// TIA Portal V20 export
FUNCTION_BLOCK "FB_ActControl"   // FB45, SCL
{ S7_Optimized_Access := 'TRUE' }
// stored: MemoryReserve 100, SetENOAutomatically false
   VAR_INPUT
      iStartSeqCond : Bool;   // Start Sequence Conditions
      iJobReq : Bool;   // Job Request - From Main
      iShuttleModeAutoPos : Bool;   // Load/Unload Manu Pos. Reached - Param
      iShuttleModeAutoPosSetPoint : LReal;   // Load/Unload Manu Pos. Setpoint - Param
      iShuttleModeSemiAutoPos : Bool;   // Load/Unload Manu Pos. Reached - Param
      iShuttleModeSemiAutoPosSetPoint : LReal;   // Load/Unload Manu Pos. Setpoint - Param
      iShuttleMoving : Bool;   // Shuttle is moving - From FB_LoaderAxis
      iShuttleInPos : Bool;   // Shuttle pos. reached - From FB_LoaderAxis
      iModeAutoPosCondition : Bool;
      iModeSemiAutoPosCondition : Bool;
      iNoStopCondition : Bool;
      iOperatorCycleRestart : Bool;
      iNC_Stopped : Bool;
      iNC_Running : Bool;
      iMissingPart : Bool;
      iExtraPart : Bool;
      iPLC_DateAndTime : DTL;
      iStepPause : Bool;
   END_VAR
   VAR_OUTPUT
      oShuttleStartReq { ExternalAccessible := 'False'; ExternalVisible := 'False'; ExternalWritable := 'False'} : Bool;   // Shuttle Start Order - To FB_LoaderAxis
      oShuttlePosSetPoint { ExternalAccessible := 'False'; ExternalVisible := 'False'; ExternalWritable := 'False'} : Real;   // Shuttle Position Setpoint - To FB_LoaderAxis
      oStopNC_Req : Bool;
      oRestartNC_Req : Bool;
      oRestartStep : Bool;
      oContinuationStep : Bool;
      oMsgMissingPart : Bool;
      oMsgExtraPart : Bool;
   END_VAR
   VAR
      sCurrent_Step_NB : Int;   // Active Step Number
      sCheck_Step_Condition : Bool;
      sOneStepForward : Bool;
      sRTOneStepForward : R_TRIG;
      sOneStepMode { S7_SetPoint := 'True'} : Bool;
      sStepForward : Bool;
      sInterface : "UDT_SequenceInterface";
      sShuttleStartReq { ExternalAccessible := 'False'; ExternalVisible := 'False'; ExternalWritable := 'False'} : Bool;
      sShuttlePosSetPoint { ExternalAccessible := 'False'; ExternalVisible := 'False'; ExternalWritable := 'False'} : Real;
      sStopNC_Req : Bool;
      sRestartNC_Req : Bool;
      sRestartStep : Bool;
      sContinuationStep : Bool;
      sMsgMissingPart : Bool;
      sMsgExtraPart : Bool;
      sHistory : Struct
         Activation : Bool;
         Steps : Array[0..99] of Int;
         Date_Time : Array[0..99] of DTL;
      END_STRUCT;
      StepText : "FB_GetTextErrorCode";
   END_VAR
   VAR_TEMP
      tIndex : Int;   // Index
   END_VAR
   VAR CONSTANT
      S00_INIT : Int := 0;
      S10_CHECK_ACT_CTRL_OPTION : Int := 10;
      S20_SHUTTLE_TO_STOP_CYCLE_POS_START_REQ : Int := 20;
      S30_SHUTTLE_TO_STOP_CYCLE_POS_REACHED : Int := 30;
      S40_STOP_CYCLE : Int := 40;
      S50_WAIT_OPERATOR_RESTART : Int := 50;
      S60_NC_RESTART : Int := 60;
      S70_UPDATE_NEXT_STEP : Int := 70;
      S120_SHUTTLE_TO_EXT_LOAD_UNLOAD_POS_START_REQ : Int := 120;
      S130_SHUTTLE_TO_EXT_LOAD_UNLOAD_POS_REACHED : Int := 130;
      S140_STOP_CYCLE : Int := 140;
      S150_WAIT_OPERATOR_RESTART : Int := 150;
      S160_NC_RESTART : Int := 160;
      S170_UPDATE_NEXT_STEP : Int := 170;
      S270_UPDATE_NEXT_STEP : Int := 270;
      S295_JOB_DONE : Int := 295;
   END_VAR
   // StepText.sCode_error[0].ErrorCode := 0;
   // StepText.sCode_error[1].ErrorCode := 10;
   // StepText.sCode_error[2].ErrorCode := 20;
   // StepText.sCode_error[3].ErrorCode := 30;
   // StepText.sCode_error[4].ErrorCode := 40;
   // StepText.sCode_error[5].ErrorCode := 50;
   // StepText.sCode_error[6].ErrorCode := 60;
   // StepText.sCode_error[7].ErrorCode := 70;
   // StepText.sCode_error[8].ErrorCode := 80;
   // StepText.sCode_error[9].ErrorCode := 90;
   // StepText.sCode_error[10].ErrorCode := 95;
BEGIN
   REGION Description header 
       //==================================================================================
       // POSALUX Swiss SA / (C) Copyright 2025
       //----------------------------------------------------------------------------------
       // Title: FB_ActControl
       // Comment/Function: 
       // Author: Fabien WALDT
       // Engineering: TIA Portal v17
       //----------------------------------------------------------------------------------
       // Change log table:
       // Version  | Date     | Expert in charge | Changes applied
       // ---------|----------|------------------|-----------------------------------------
       // 00.00.01 | 20250527 | WFA              | First released version
       // =================================================================================
   END_REGION

   REGION Define condition to start
       IF #iStartSeqCond THEN
           #sInterface.SequenceReleased := TRUE;
       ELSE
           // Standard sequencer controls
           #sInterface.SequenceReleased := FALSE;
           #sCurrent_Step_NB := #S00_INIT;
           #sInterface.SequenceRun := FALSE;
           #sInterface.JobDone := FALSE;
           #sCheck_Step_Condition := FALSE;

           // Dedicated sequencer controls
           #sShuttleStartReq := FALSE;
           #sShuttlePosSetPoint := 0.0;
           #sStopNC_Req := FALSE;
           #sRestartNC_Req := FALSE;
           #sRestartStep := FALSE;
           #sContinuationStep := FALSE;


           // Add specifics controls 
       END_IF;

       // Reset interface error
       IF #sInterface.Reset THEN
           #sInterface.Error := FALSE;
       END_IF;

       // Reset start when axis in position
       IF #iShuttleInPos THEN
           #sShuttleStartReq := FALSE;
       END_IF;

       // One step forward
       #sRTOneStepForward.CLK := #sOneStepForward;
       #sRTOneStepForward();
       #sStepForward := (NOT #sOneStepMode OR (#sOneStepMode AND #sRTOneStepForward.Q)) AND NOT #iStepPause;
       #sOneStepForward := FALSE;

       // Action only true in dedicated steps
       #sStopNC_Req := FALSE;
       #sRestartNC_Req := FALSE;
   END_REGION

   REGION Sequence Function
       CASE #sCurrent_Step_NB OF
           #S00_INIT:
               REGION S00 INIT
                   #sCheck_Step_Condition := TRUE;
                   #sMsgMissingPart := FALSE;
                   #sMsgExtraPart := FALSE;
               END_REGION
           #S10_CHECK_ACT_CTRL_OPTION:
               REGION S10_CHECK_ACT_CTRL_OPTION
                   #sCheck_Step_Condition := TRUE;
               END_REGION
           #S20_SHUTTLE_TO_STOP_CYCLE_POS_START_REQ:
               REGION S20_SHUTTLE_TO_STOP_CYCLE_POS_START_REQ
                   #sShuttleStartReq := NOT #iShuttleModeAutoPos;
                   #sShuttlePosSetPoint := LREAL_TO_REAL(#iShuttleModeAutoPosSetPoint);
                   #sCheck_Step_Condition := TRUE;
               END_REGION
           #S30_SHUTTLE_TO_STOP_CYCLE_POS_REACHED:
               REGION S30_SHUTTLE_TO_STOP_CYCLE_POS_REACHED
                   #sCheck_Step_Condition := TRUE;
               END_REGION
           #S40_STOP_CYCLE:
               REGION S40_STOP_CYCLE
                   #sStopNC_Req := TRUE;
                   #sMsgMissingPart := #iMissingPart;
                   #sMsgExtraPart := #iExtraPart;
                   #sCheck_Step_Condition := TRUE;
               END_REGION
           #S50_WAIT_OPERATOR_RESTART:
               REGION S50_WAIT_OPERATOR_RESTART
                   #sCheck_Step_Condition := TRUE;
               END_REGION
           #S60_NC_RESTART:
               REGION S60_NC_RESTART
                   #sRestartNC_Req := TRUE;
                   #sCheck_Step_Condition := TRUE;
               END_REGION
           #S70_UPDATE_NEXT_STEP:
               REGION S70_UPDATE_NEXT_STEP
                   #sRestartStep := TRUE;
                   #sContinuationStep := FALSE;
                   #sCheck_Step_Condition := TRUE;
               END_REGION

           #S120_SHUTTLE_TO_EXT_LOAD_UNLOAD_POS_START_REQ:
               REGION S120_SHUTTLE_TO_EXT_LOAD_UNLOAD_POS_START_REQ
                   #sShuttleStartReq := NOT #iShuttleModeSemiAutoPos;
                   #sShuttlePosSetPoint := LREAL_TO_REAL(#iShuttleModeSemiAutoPosSetPoint);
                   #sCheck_Step_Condition := TRUE;
               END_REGION
           #S130_SHUTTLE_TO_EXT_LOAD_UNLOAD_POS_REACHED:
               REGION S130_SHUTTLE_TO_EXT_LOAD_UNLOAD_POS_REACHED
                   #sCheck_Step_Condition := TRUE;
               END_REGION
           #S140_STOP_CYCLE:
               REGION S140_STOP_CYCLE
                   #sStopNC_Req := TRUE;
                   #sMsgMissingPart := #iMissingPart;
                   #sMsgExtraPart := #iExtraPart;
                   #sCheck_Step_Condition := TRUE;
               END_REGION
           #S150_WAIT_OPERATOR_RESTART:
               REGION S150_WAIT_OPERATOR_RESTART
                   #sCheck_Step_Condition := TRUE;
               END_REGION
           #S160_NC_RESTART:
               REGION S160_NC_RESTART
                   #sRestartNC_Req := TRUE;
                   #sCheck_Step_Condition := TRUE;
               END_REGION
           #S170_UPDATE_NEXT_STEP:
               REGION S170_UPDATE_NEXT_STEP
                   #sRestartStep := TRUE;
                   #sContinuationStep := FALSE;
                   #sCheck_Step_Condition := TRUE;
               END_REGION

           #S270_UPDATE_NEXT_STEP:
               REGION S270_UPDATE_NEXT_STEP
                   #sRestartStep := FALSE;
                   #sContinuationStep := TRUE;
                   #sCheck_Step_Condition := TRUE;
               END_REGION

           #S295_JOB_DONE:
               REGION S295_JOB_DONE
                   #sInterface.JobDone := TRUE;
                   #sCheck_Step_Condition := TRUE;
               END_REGION
           ELSE:
               #sInterface.Error := TRUE;
       END_CASE;
   END_REGION

   REGION Sequence Next Step Condition
       IF #sCheck_Step_Condition THEN
           CASE #sCurrent_Step_NB OF
               #S00_INIT:
                   REGION S00 INIT
                       IF #sInterface.SequenceReleased AND #iJobReq THEN
                           #sCurrent_Step_NB := #S10_CHECK_ACT_CTRL_OPTION;
                           #sInterface.SequenceRun := TRUE;
                           #sCheck_Step_Condition := FALSE;
                       ELSE
                           #sInterface.SequenceRun := FALSE;
                       END_IF;
                   END_REGION
               #S10_CHECK_ACT_CTRL_OPTION:
                   REGION S10_CHECK_ACT_CTRL_OPTION
                       IF #sInterface.SequenceReleased AND #sStepForward AND #iModeAutoPosCondition AND NOT #iModeSemiAutoPosCondition AND NOT #iNoStopCondition THEN
                           #sCurrent_Step_NB := #S20_SHUTTLE_TO_STOP_CYCLE_POS_START_REQ;
                           #sCheck_Step_Condition := FALSE;
                       ELSIF #sInterface.SequenceReleased AND #sStepForward AND NOT #iModeAutoPosCondition AND #iModeSemiAutoPosCondition AND NOT #iNoStopCondition THEN
                           #sCurrent_Step_NB := #S120_SHUTTLE_TO_EXT_LOAD_UNLOAD_POS_START_REQ;
                           #sCheck_Step_Condition := FALSE;
                       ELSIF #sInterface.SequenceReleased AND #sStepForward AND NOT #iModeAutoPosCondition AND NOT #iModeSemiAutoPosCondition AND #iNoStopCondition THEN
                           #sCurrent_Step_NB := #S270_UPDATE_NEXT_STEP;
                           #sCheck_Step_Condition := FALSE;
                       END_IF;
                   END_REGION
               #S20_SHUTTLE_TO_STOP_CYCLE_POS_START_REQ:
                   REGION S20_SHUTTLE_TO_STOP_CYCLE_POS_START_REQ
                       IF #sInterface.SequenceReleased AND #sStepForward AND (#iShuttleMoving OR #iShuttleModeAutoPos) THEN
                           #sCurrent_Step_NB := #S30_SHUTTLE_TO_STOP_CYCLE_POS_REACHED;
                           #sCheck_Step_Condition := FALSE;
                       END_IF;
                   END_REGION
               #S30_SHUTTLE_TO_STOP_CYCLE_POS_REACHED:
                   REGION S30_SHUTTLE_TO_STOP_CYCLE_POS_REACHED
                       IF #sInterface.SequenceReleased AND #sStepForward AND NOT #sShuttleStartReq AND #iShuttleModeAutoPos THEN
                           #sCurrent_Step_NB := #S40_STOP_CYCLE;
                           #sCheck_Step_Condition := FALSE;
                       END_IF;
                   END_REGION
               #S40_STOP_CYCLE:
                   REGION S40_STOP_CYCLE
                       IF #sInterface.SequenceReleased AND #sStepForward AND #iNC_Stopped THEN
                           #sCurrent_Step_NB := #S50_WAIT_OPERATOR_RESTART;
                           #sCheck_Step_Condition := FALSE;
                       END_IF;
                   END_REGION
                   #S50_WAIT_OPERATOR_RESTART:
                       REGION S50_WAIT_OPERATOR_RESTART
                           IF #sInterface.SequenceReleased AND #sStepForward AND #iOperatorCycleRestart THEN
                               #sCurrent_Step_NB := #S60_NC_RESTART;
                               #sCheck_Step_Condition := FALSE;
                           END_IF;
                       END_REGION
                   #S60_NC_RESTART:
                       REGION S60_NC_RESTART
                           IF #sInterface.SequenceReleased AND #sStepForward AND #iNC_Running THEN
                               #sCurrent_Step_NB := #S70_UPDATE_NEXT_STEP;
                               #sCheck_Step_Condition := FALSE;
                           END_IF;
                       END_REGION
                   #S70_UPDATE_NEXT_STEP:
                       REGION S70_UPDATE_NEXT_STEP
                           IF #sInterface.SequenceReleased AND #sStepForward AND "AlwaysTRUE" THEN
                               #sCurrent_Step_NB := #S295_JOB_DONE;
                               #sCheck_Step_Condition := FALSE;
                           END_IF;
                       END_REGION

                   #S120_SHUTTLE_TO_EXT_LOAD_UNLOAD_POS_START_REQ:
                       REGION S120_SHUTTLE_TO_EXT_LOAD_UNLOAD_POS_START_REQ
                           IF #sInterface.SequenceReleased AND #sStepForward AND (#iShuttleMoving OR #iShuttleModeSemiAutoPos) THEN
                               #sCurrent_Step_NB := #S130_SHUTTLE_TO_EXT_LOAD_UNLOAD_POS_REACHED;
                               #sCheck_Step_Condition := FALSE;
                           END_IF;
                       END_REGION
                   #S130_SHUTTLE_TO_EXT_LOAD_UNLOAD_POS_REACHED:
                       REGION S130_SHUTTLE_TO_EXT_LOAD_UNLOAD_POS_REACHED
                           IF #sInterface.SequenceReleased AND #sStepForward AND NOT #sShuttleStartReq AND #iShuttleModeSemiAutoPos THEN
                               #sCurrent_Step_NB := #S140_STOP_CYCLE;
                               #sCheck_Step_Condition := FALSE;
                           END_IF;
                       END_REGION
                   #S140_STOP_CYCLE:
                       REGION S140_STOP_CYCLE
                           IF #sInterface.SequenceReleased AND #sStepForward AND #iNC_Stopped THEN
                               #sCurrent_Step_NB := #S150_WAIT_OPERATOR_RESTART;
                               #sCheck_Step_Condition := FALSE;
                           END_IF;
                       END_REGION
                       #S150_WAIT_OPERATOR_RESTART:
                           REGION S150_EXCHANGE_EXT_LOADER_IN_PROGRESS
                               IF #sInterface.SequenceReleased AND #sStepForward AND #iOperatorCycleRestart THEN
                                   #sCurrent_Step_NB := #S160_NC_RESTART;
                                   #sCheck_Step_Condition := FALSE;
                               END_IF;
                           END_REGION
                       #S160_NC_RESTART:
                           REGION S60_NC_RESTART
                               IF #sInterface.SequenceReleased AND #sStepForward AND #iNC_Running THEN
                                   #sCurrent_Step_NB := #S170_UPDATE_NEXT_STEP;
                                   #sCheck_Step_Condition := FALSE;
                               END_IF;
                           END_REGION
                       #S170_UPDATE_NEXT_STEP:
                           REGION S70_UPDATE_NEXT_STEP
                               IF #sInterface.SequenceReleased AND #sStepForward AND "AlwaysTRUE" THEN
                                   #sCurrent_Step_NB := #S295_JOB_DONE;
                                   #sCheck_Step_Condition := FALSE;
                               END_IF;
                           END_REGION
                       #S270_UPDATE_NEXT_STEP:
                           REGION S270_UPDATE_NEXT_STEP
                               IF #sInterface.SequenceReleased AND #sStepForward AND "AlwaysTRUE" THEN
                                   #sCurrent_Step_NB := #S295_JOB_DONE;
                                   #sCheck_Step_Condition := FALSE;
                               END_IF;
                           END_REGION
                       #S295_JOB_DONE:
                           REGION S295_JOB_DONE
                               IF NOT #iJobReq THEN
                                   #sCurrent_Step_NB := #S00_INIT;
                                   #sCheck_Step_Condition := FALSE;
                                   #sInterface.JobDone := FALSE;
                               END_IF;
                           END_REGION
               ELSE
                   #sInterface.Error := TRUE;
           END_CASE;
       END_IF;
   END_REGION

   REGION Outputs Update
       #oShuttleStartReq := #sShuttleStartReq;
       #oShuttlePosSetPoint := #sShuttlePosSetPoint;
       #oStopNC_Req := #sStopNC_Req;
       #oRestartNC_Req := #sRestartNC_Req;
       #oRestartStep := #sRestartStep;
       #oContinuationStep := #sContinuationStep;
       #oMsgMissingPart := #sMsgMissingPart;
       #oMsgExtraPart := #sMsgExtraPart;
   END_REGION

   REGION Steps - Date and Time History
       IF #sHistory.Activation THEN
           IF #sHistory.Steps[0] <> #sCurrent_Step_NB THEN
               FOR #tIndex := 98 TO 0 BY -1 DO
                   #sHistory.Steps[#tIndex + 1] := #sHistory.Steps[#tIndex];
                   #sHistory.Date_Time[#tIndex + 1] := #sHistory.Date_Time[#tIndex];
               END_FOR;
               #sHistory.Steps[0] := #sCurrent_Step_NB;
               #sHistory.Date_Time[0] := #iPLC_DateAndTime;
           END_IF;
       END_IF;
   END_REGION

   REGION Steps Text
       #StepText(iErrorCode := #sCurrent_Step_NB,
                 oErrorText => #StepText.oErrorText);
   END_REGION
END_FUNCTION_BLOCK
